FUNCTION F_ComputeFixed64Size : UDINT
VAR_INPUT
    {attribute 'analysis' := '-33' }
    nValue : ULINT;
END_VAR


F_ComputeFixed64Size := GCL_PB.cLittleEndian64Size;

END_FUNCTION

(* stored: Version 1.1.0.1
   POU F_ComputeFixed64Size: Id {e5e4f583-643e-4c6c-a551-2106e84f4e70}, SpecialFunc None *)
